// TIA Portal V20 export
TYPE "LConSMC_typeSectionalDriveConfig"
// Konfigurationsdaten der Bahnzugregelung / Configuration data of the sectional drive
// stored: Access Published
   STRUCT
      positionControlled : Bool := FALSE;   // TRUE: Achse wird lagegeregelt betrieben FALSE: Achse wird Drehzahlgeregelt betrieben / TRUE: Enable MoveVelocity position controlled in case of positioning axis
      axisCtrl : Bool := TRUE;   // TRUE: Sollwerte werden an den Antrieb gesendet FALSE: Es werden nur Sollwerte berechnet aber es erfolgt keine Kommunikation mit dem Antrieb / FALSE: No axis control just calculated setpoints TRUE: Use MoveVelocity to forward setpoints to axis
      jogVelocity : Real;   // [m/min oder ft/min] Bahngeschwindigkeit zum Vertippen der Achse über die Eingänge "jogPos" und "jogNeg" / [m/min oder ft/min] Web velocity to jog the drive via the inputs "jogPos" and "jogNeg"
      diameter : LReal := 1.0;   // [m oder inch] Durchmesser der Zugwalze / [m or inch] Diameter of sectional drive axis
      overrideVelocity : Real := 10.0;   // [m/min oder ft/min] Additive Zusatzgeschwindigkeit zur Übersteuerung des Drehzahlreglers. Dieser Wer wird in den drehmomentengeregelten Modi benötigt (controlMode = 1-3) / [m/min or ft/min] Additive velocity offset for speed controller This value is only needed for the torque controlled modes (controlMode = 1-3)
      maxVelocity : Real := 0.0;   // [m/min or ft/min] Maximum possible web velocity. Maximum speed setpoint of the axis is limited to maxVelocity (+ overrideVelocity) and minimum diameter
      getAxisConfigAtStart : Bool := TRUE;   // TRUE: Achskonfiguration (Getriebe, Referenzdrehmoment, Achseinheiten) wird mit steigender Flanke an "enable" ausgelesen FALSE: Die Konfigurationsdaten müssen manuell in der Konfigurationsstruktur eingegeben werden / TRUE: Readout gear,reference torque and units from axis with rising edge. FALSE: Take config values
      noOfSamplesLineVelocity : UInt := 1;   // Anzahl an samples für die gleitende Mittelwertbildung des Bahnsollwertes während dem Aufsynchronisieren auf eine fahrende Bahn / Number of samples for moving average filter of line velocity setpoint for synchronizing to a moving web
      unitConfiguration { S7_SetPoint := 'True'} : "LConSMC_typeUnitConfiguration";   // Konfiguration der Einheiten / Configuration of the units
      SectionalDriveDynamics { S7_SetPoint := 'True'} : "LConSMC_typeAxisDynamics";   // Konfiguration der Dynamiken / Configuration of the axis dynamics
      technologyControllerConfig { S7_SetPoint := 'True'} : "LConSMC_typeTechnologyControllerConfig";   // Konfiguration des Technologiereglers (Tänzer oder Zugmessdose) / Configuration parameters for technology controller (Dancer or load cell)
      torquePrecontrolConfig { S7_SetPoint := 'True'} : "LConSMC_typeSectionalDriveTorquePrecontrolConfig";   // Konfiguration der Drehmomentenvorsteuerung / Configuration parameters for torque precontrol
      webbreakDetectionConfig { S7_SetPoint := 'True'} : "LConSMC_typeWebbreakDetectConfig";   // Konfiguration der Bahnrisserkennung / Configuration parameters for webbreak detection
   END_STRUCT;
END_TYPE
